// TIA Portal V20 export
FUNCTION_BLOCK "BlowOffValve"   // FB550, FBD
{ S7_Optimized_Access := 'TRUE' }
// stored: AutoNumber false, MemoryReserve 100, SetENOAutomatically false
   VAR
      Var { ExternalAccessible := 'False'; ExternalVisible := 'False'; ExternalWritable := 'False'} : "TypeVar";
      T { ExternalAccessible := 'False'; ExternalVisible := 'False'; ExternalWritable := 'False'} : Array[1..20] of IEC_TIMER;
      blowOff { ExternalAccessible := 'False'; ExternalVisible := 'False'; ExternalWritable := 'False'} : Bool;
      breakTime { ExternalAccessible := 'False'; ExternalVisible := 'False'; ExternalWritable := 'False'} : Time;
      intervallTime { ExternalAccessible := 'False'; ExternalVisible := 'False'; ExternalWritable := 'False'} : Time;
      intervallTimeOff { ExternalAccessible := 'False'; ExternalVisible := 'False'; ExternalWritable := 'False'} : Time;
      bottom { ExternalAccessible := 'False'; ExternalVisible := 'False'; ExternalWritable := 'False'} : Struct
         delayStart : Time;
         Impuls : Time;
         start : Bool;
         blowOff : Bool;
      END_STRUCT;
      left { ExternalAccessible := 'False'; ExternalVisible := 'False'; ExternalWritable := 'False'} : Struct
         delayStart : Time;
         Impuls : Time;
         start : Bool;
         blowOff : Bool;
      END_STRUCT;
      right { ExternalAccessible := 'False'; ExternalVisible := 'False'; ExternalWritable := 'False'} : Struct
         delayStart : Time;
         Impuls : Time;
         start : Bool;
         blowOff : Bool;
      END_STRUCT;
      xray { ExternalAccessible := 'False'; ExternalVisible := 'False'; ExternalWritable := 'False'} : Struct
         delayStart : Time;
         Impuls : Time;
         start : Bool;
         blowOff : Bool;
      END_STRUCT;
   END_VAR
   VAR_TEMP   // added for the SCL form of the ladder/FBD networks
      _w1 : Bool;
   END_VAR
BEGIN

REGION Network 1: pneumatic ok
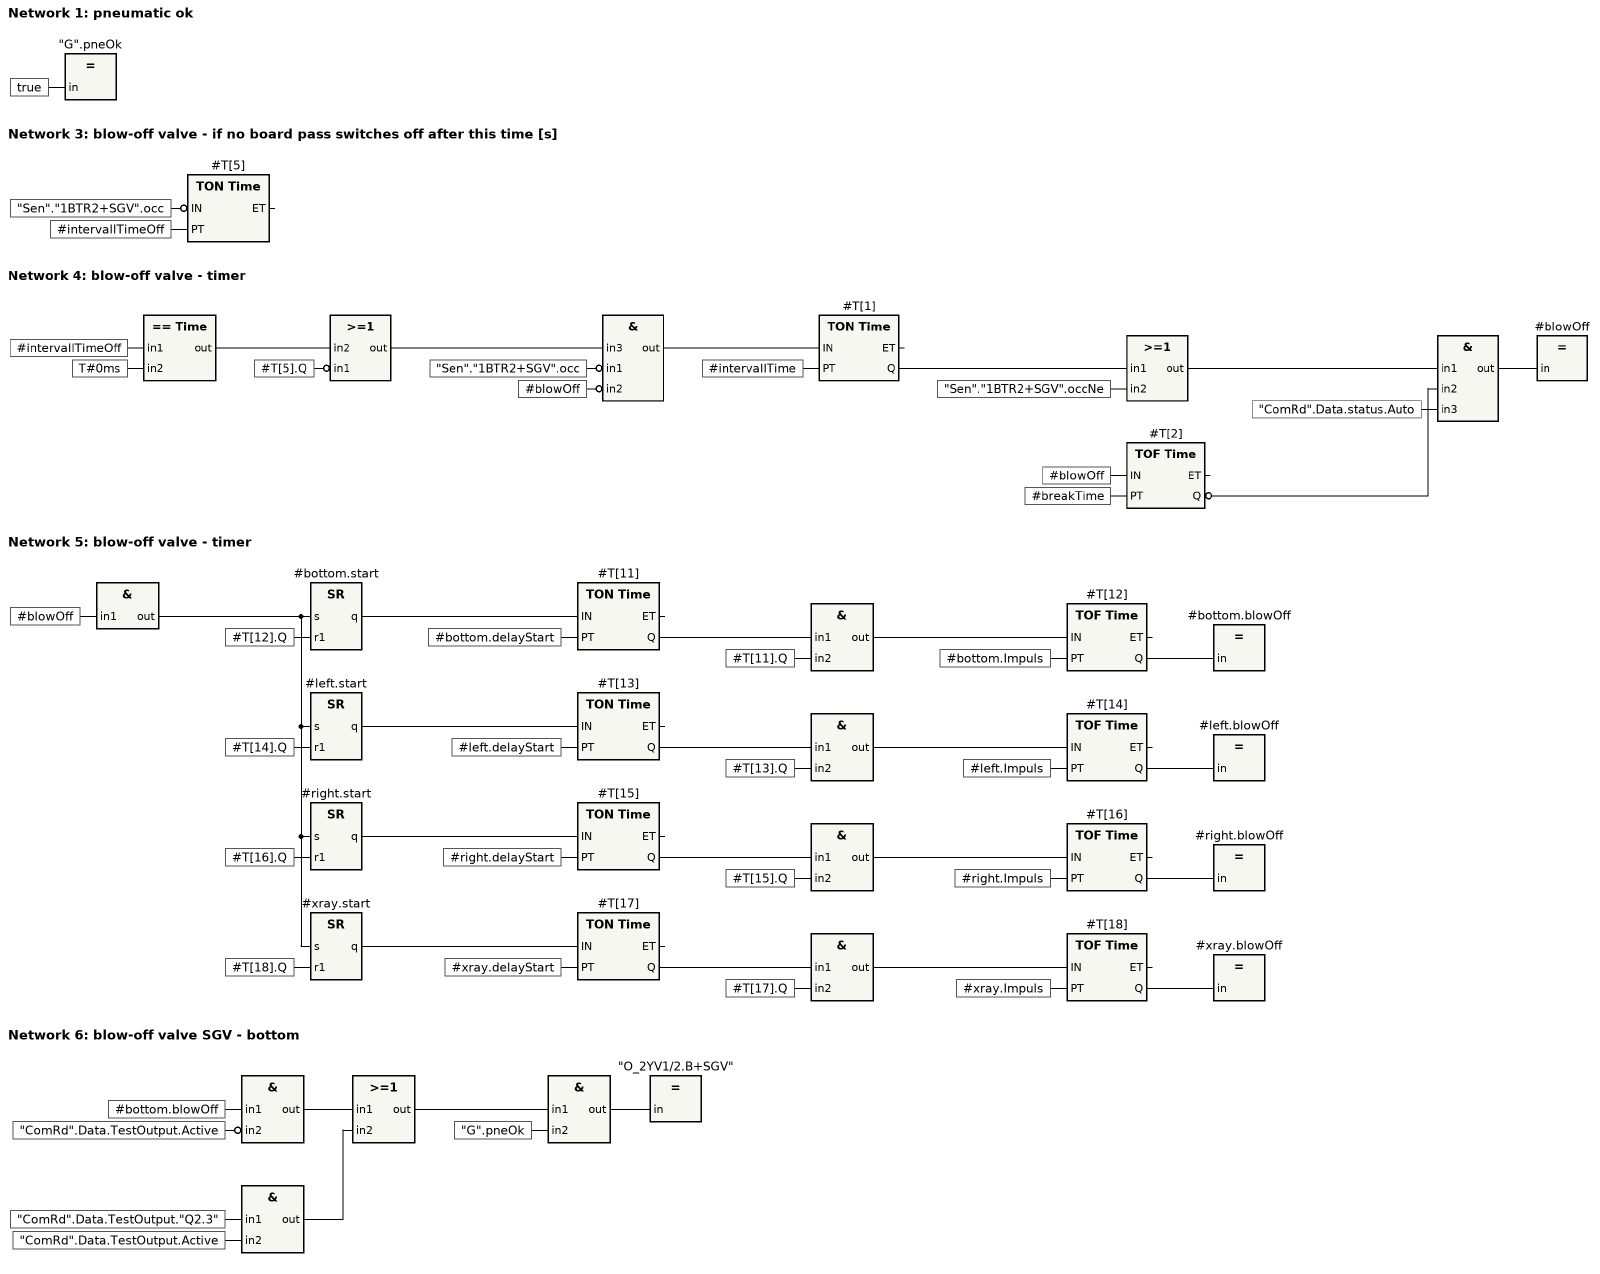
   "G".pneOk := true;
END_REGION

REGION Network 2 (SCL): blow-off valve - parameter

   #breakTime := INT_TO_TIME("Param".Rd.blowOffIbreak);
   #intervallTime := UDINT_TO_TIME(INT_TO_UDINT("Param".Rd.blowOffintervall) * 1000);
   #intervallTimeOff := UDINT_TO_TIME(INT_TO_UDINT("Param".Rd.blowOffintervallOff) * 1000);

   // bottom
   #bottom.delayStart := INT_TO_TIME("Param".Rd.blowOffDelayStartBottom);
   IF "Param".Rd.blowOffImpulsBottom <> 0 THEN
       #bottom.Impuls := INT_TO_TIME("Param".Rd.blowOffImpulsBottom);
   ELSE
       #bottom.Impuls := INT_TO_TIME("Param".Rd.blowOffImpuls);
   END_IF;

   // left
   #left.delayStart := INT_TO_TIME("Param".Rd.blowOffDelayStartLeft);
   IF "Param".Rd.blowOffImpulsLeft <> 0 THEN
       #left.Impuls := INT_TO_TIME("Param".Rd.blowOffImpulsLeft);
   ELSE
       #left.Impuls := INT_TO_TIME("Param".Rd.blowOffImpuls);
   END_IF;

   // right
   #right.delayStart := INT_TO_TIME("Param".Rd.blowOffDelayStartRight);
   IF "Param".Rd.blowOffImpulsRight <> 0 THEN
       #right.Impuls := INT_TO_TIME("Param".Rd.blowOffImpulsRight);
   ELSE
       #right.Impuls := INT_TO_TIME("Param".Rd.blowOffImpuls);
   END_IF;

   // xray
   #xray.delayStart := INT_TO_TIME("Param".Rd.blowOffDelayStartXray);
   IF "Param".Rd.blowOffImpulsXray <> 0 THEN
       #xray.Impuls := INT_TO_TIME("Param".Rd.blowOffImpulsXray);
   ELSE
       #xray.Impuls := INT_TO_TIME("Param".Rd.blowOffImpuls);
   END_IF;
END_REGION

REGION Network 3: blow-off valve - if no board pass switches off after this time [s]
   #T[5].TON(IN := NOT "Sen"."1BTR2+SGV".occ, PT := #intervallTimeOff);
END_REGION

REGION Network 4: blow-off valve - timer
   #T[1].TON(IN := ((#intervallTimeOff = T#0ms) OR NOT #T[5].Q) AND NOT "Sen"."1BTR2+SGV".occ AND NOT #blowOff,
             PT := #intervallTime);
   #_w1 := #T[1].Q OR "Sen"."1BTR2+SGV".occNe;
   #T[2].TOF(IN := #blowOff, PT := #breakTime);
   #blowOff := #_w1 AND NOT #T[2].Q AND "ComRd".Data.status.Auto;
END_REGION

REGION Network 5: blow-off valve - timer
   IF #blowOff THEN
       #bottom.start := TRUE;   // SR flip-flop
   END_IF;
   IF #T[12].Q THEN #bottom.start := FALSE; END_IF;
   #T[11].TON(IN := #bottom.start, PT := #bottom.delayStart);
   #T[12].TOF(IN := #T[11].Q AND #T[11].Q, PT := #bottom.Impuls);
   #bottom.blowOff := #T[12].Q;
   IF #blowOff THEN
       #left.start := TRUE;   // SR flip-flop
   END_IF;
   IF #T[14].Q THEN #left.start := FALSE; END_IF;
   #T[13].TON(IN := #left.start, PT := #left.delayStart);
   #T[14].TOF(IN := #T[13].Q AND #T[13].Q, PT := #left.Impuls);
   #left.blowOff := #T[14].Q;
   IF #blowOff THEN
       #right.start := TRUE;   // SR flip-flop
   END_IF;
   IF #T[16].Q THEN #right.start := FALSE; END_IF;
   #T[15].TON(IN := #right.start, PT := #right.delayStart);
   #T[16].TOF(IN := #T[15].Q AND #T[15].Q, PT := #right.Impuls);
   #right.blowOff := #T[16].Q;
   IF #blowOff THEN
       #xray.start := TRUE;   // SR flip-flop
   END_IF;
   IF #T[18].Q THEN #xray.start := FALSE; END_IF;
   #T[17].TON(IN := #xray.start, PT := #xray.delayStart);
   #T[18].TOF(IN := #T[17].Q AND #T[17].Q, PT := #xray.Impuls);
   #xray.blowOff := #T[18].Q;
END_REGION

REGION Network 6: blow-off valve SGV - bottom
   "O_2YV1/2.B+SGV" := ((#bottom.blowOff AND NOT "ComRd".Data.TestOutput.Active) OR ("ComRd".Data.TestOutput."Q2.3" AND "ComRd".Data.TestOutput.Active)) AND "G".pneOk;
END_REGION

REGION Network 7: blow-off valve SGV - left
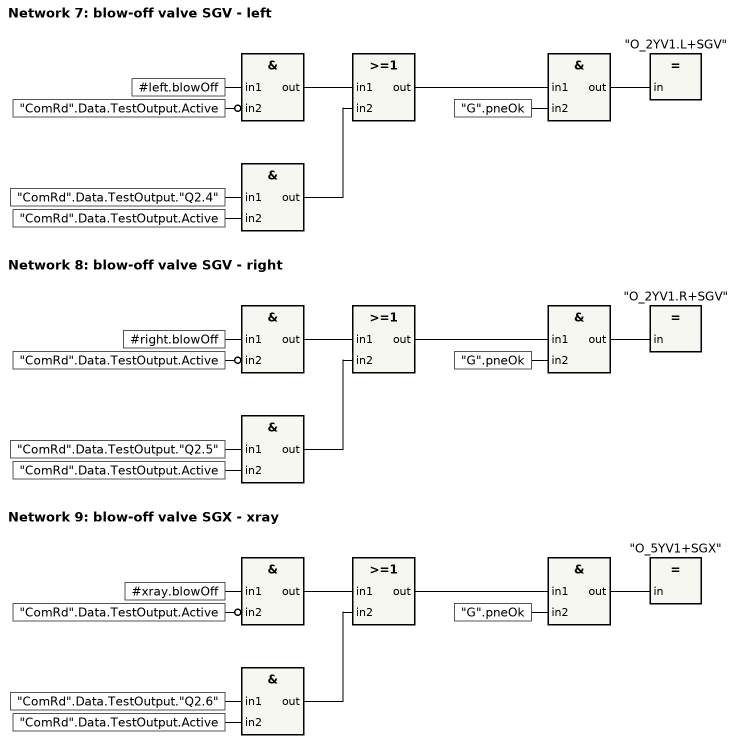
   "O_2YV1.L+SGV" := ((#left.blowOff AND NOT "ComRd".Data.TestOutput.Active) OR ("ComRd".Data.TestOutput."Q2.4" AND "ComRd".Data.TestOutput.Active)) AND "G".pneOk;
END_REGION

REGION Network 8: blow-off valve SGV - right
   "O_2YV1.R+SGV" := ((#right.blowOff AND NOT "ComRd".Data.TestOutput.Active) OR ("ComRd".Data.TestOutput."Q2.5" AND "ComRd".Data.TestOutput.Active)) AND "G".pneOk;
END_REGION

REGION Network 9: blow-off valve SGX - xray
   "O_5YV1+SGX" := ((#xray.blowOff AND NOT "ComRd".Data.TestOutput.Active) OR ("ComRd".Data.TestOutput."Q2.6" AND "ComRd".Data.TestOutput.Active)) AND "G".pneOk;
END_REGION
END_FUNCTION_BLOCK
